FUNCTION_BLOCK ControlHMI (* Composite Function Block Type *)
  (* Standard: 61499-2 *)
  (* Version 0.0, 23/09/2021, Pranay Jhunjhunwala, Schneider Electric, template *)
  PACKAGE Main;
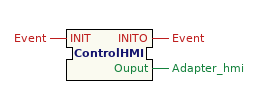
  EVENT_INPUT
    INIT; (* Initialization Request *)
  END_EVENT
  EVENT_OUTPUT
    INITO; (* Initialization Confirm *)
  END_EVENT
  PLUGS
    Ouput : Adapter_hmi;
  END_PLUGS
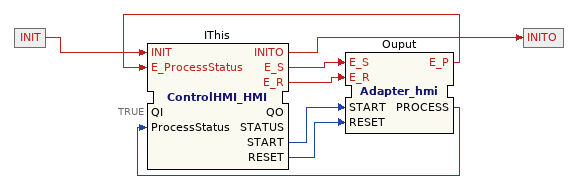
  FBS
    IThis : ControlHMI_HMI(QI := TRUE);
  END_FBS
  EVENT_CONNECTIONS
    INIT TO IThis.INIT;
    Ouput.E_P TO IThis.E_ProcessStatus;
    IThis.INITO TO INITO;
    IThis.E_S TO Ouput.E_S;
    IThis.E_R TO Ouput.E_R;
  END_CONNECTIONS
  DATA_CONNECTIONS
    Ouput.PROCESS TO IThis.ProcessStatus;
    IThis.START TO Ouput.START;
    IThis.RESET TO Ouput.RESET;
  END_CONNECTIONS
END_FUNCTION_BLOCK
